(* CODESYS project IO Link.library
   Company: Ziga Javornik
   DefaultNamespace: ZigaLibs.IoLink
   Version: 0.0.0.1
   Placeholder: ZigaLibs.IoLink
   Author: Ziga Javornik
   Description: IO link implementaiton libray
   Title: ZigaLibs.IoLink

Project tree, tasks and I/O mapping:
  libraries: Tc2_Standard, * (Beckhoff Automation GmbH); Tc2_System, * (Beckhoff Automation GmbH); Tc3_Module, * (Beckhoff Automation GmbH); TcUnit, * (www.tcunit.org); ZigaLibs.Logging, 0.0.4.1 (Ziga Javornik)
  GVLs/
  SOURCE/
    function block FB_IoLinkChannel_64Byte [ST]
    function block FB_IoLinkState [ST]: ChannelState, FB_init, GetChannelState
    data type ST_IoLink_ChannelState
    data type T_IoLink64ByteData
  TESTS/
    Test suites/
      function block FB_SUT_Tests [ST]: TestXX_Template
    program PRG_TESTS [ST]
*)

// SOURCE/ST_IoLink_ChannelState
{attribute 'qualified_only'}
{attribute 'strict'}
{attribute 'to_string'}
TYPE ST_IoLink_ChannelState :
STRUCT
	PortDisabled 				: BOOL;
	PortInStdDigIn 				: BOOL;
	PortInStdDigOut				: BOOL;
	PortInCommunicationOP		: BOOL;
	PortInCommunicationCOMSTOP	: BOOL;
	WatchdogDetected			: BOOL;
	InternalError				: BOOL;
	InvalidDeviceId				: BOOL;
	InvalidVendorId				: BOOL;
	InvalidIoLinkVersion		: BOOL;
	InvalidFrameCapability		: BOOL;
	InvalidCycleTime			: BOOL;
	InvalidPD_InLength			: BOOL;
	InvalidPD_OutLength			: BOOL;
	NoDeviceDetected			: BOOL;
	ErrorPreoperate				: BOOL;
END_STRUCT
END_TYPE

// SOURCE/T_IoLink64ByteData
TYPE 
	T_IoLink64ByteData : ARRAY[0..7] OF BYTE; 
END_TYPE

// SOURCE/FB_IoLinkChannel_64Byte
FUNCTION_BLOCK ABSTRACT FB_IoLinkChannel_64Byte
VAR_INPUT
END_VAR
VAR_OUTPUT
END_VAR
VAR
	Inputs 	AT %I*	: T_IoLink64ByteData;
	Outputs	AT %Q*	: T_IoLink64ByteData;
END_VAR

END_FUNCTION_BLOCK

// SOURCE/FB_IoLinkState
FUNCTION_BLOCK ABSTRACT FB_IoLinkState
VAR_INPUT
END_VAR
VAR_OUTPUT
END_VAR
VAR
	State	 AT%I*	: USINT;
	_channelState 	: ST_IoLink_ChannelState;
	_logger			: REFERENCE TO ZigaLibs_Logging.I_Logger;
END_VAR

 {attribute 'monitoring' := 'variable'}
// Gets the IO link channel state info
PROPERTY PUBLIC ChannelState : REFERENCE TO ST_IoLink_ChannelState
GET
_channelState := THIS^.GetChannelState();
ChannelState REF= _channelState;
END_GET
END_PROPERTY

METHOD FB_init : BOOL
VAR_INPUT
	bInitRetains : BOOL; // if TRUE, the retain variables are initialized (warm start / cold start)
	bInCopyCode : BOOL;  // if TRUE, the instance afterwards gets moved into the copy code (online change)
	logger			: REFERENCE TO ZigaLibs_Logging.I_Logger;
END_VAR
_logger REF= logger;
END_METHOD

// Gets the channel state based on the State value transfered from the hardware device
METHOD PUBLIC GetChannelState : ST_IoLink_ChannelState

VAR
	nMaskedState	: USINT;
	result			: ST_IoLink_ChannelState;
END_VAR
nMaskedState := 16#0F AND THIS^.State;
result.PortDisabled := nMaskedState = 16#00;
result.PortInStdDigIn := nMaskedState = 16#01;
result.PortInStdDigOut := nMaskedState = 16#02;
result.PortInCommunicationOP := nMaskedState = 16#03;
result.PortInCommunicationCOMSTOP := nMaskedState = 16#04;

nMaskedState := 16#F0 AND THIS^.State;
result.WatchdogDetected := nMaskedState = 16#10;
result.InternalError := nMaskedState = 16#20;
result.InvalidDeviceId := nMaskedState = 16#30;
result.InvalidVendorId := nMaskedState = 16#40;
result.InvalidIoLinkVersion := nMaskedState = 16#50;
result.InvalidFrameCapability := nMaskedState = 16#60;
result.InvalidCycleTime := nMaskedState = 16#70;
result.InvalidPD_InLength := nMaskedState = 16#80;
result.InvalidPD_OutLength := nMaskedState = 16#90;
result.NoDeviceDetected := nMaskedState = 16#A0;
result.ErrorPreoperate := nMaskedState = 16#B0;

GetChannelState := result;
END_METHOD

END_FUNCTION_BLOCK

// TESTS/Test suites/FB_SUT_Tests
// Subject under test
FUNCTION_BLOCK FB_SUT_Tests EXTENDS FB_TestSuite

// Create instance variables that will be accesible for all tests
VAR
END_VAR

// Call your test methods here
TestXX_Template();

METHOD PRIVATE TestXX_Template

(* Instanced variables are VERY useful for writing tests since tests are run in paralel (by default).
By instantiating local variables that are not placed on the same stack as method (values are retained between calls)
you make sure that the SUT is not changed by some other test. *)
VAR_INST
	
END_VAR

// Place temporary variables here
VAR
	
END_VAR
// The name of the test, is the same as method name!
// Use this for paralel unit tests
// TcUnit.TEST('TestXX_Template');

// Use this for running tests in sequence
IF TcUnit.TEST_ORDERED('TestXX_Template') THEN
	// Do your assertions here...
	AssertTrue(
		Condition := FALSE, 
		Message := 'Implement tests!');

	TcUnit.TEST_FINISHED();
END_IF
END_METHOD

END_FUNCTION_BLOCK

// TESTS/PRG_TESTS
PROGRAM PRG_TESTS

(* Instantiate test suites here. Naming convention for tests should be a suffix with _Tests.
Good practice for creating test methods is to end them with _test as well. *)
VAR
	fbSUT_Tests	: FB_SUT_Tests;
END_VAR

// Run tests in parallel
//TcUnit.RUN();

// Run tests in sequence, one after the other.
TcUnit.RUN_IN_SEQUENCE();

END_PROGRAM
